{attribute 'qualified_only'}
VAR_GLOBAL
	MyFub : TestFub;
	MyStruct: TestStructure; 	
END_VAR

(* stored: Version 1.1.0.1, ProductVersion 3.1.4024.12
   GVL GVL: Id {0048069a-d4d8-486e-aafb-7576e6aaa7d9} *)
